TEXTLIST TL_E_CTRL_XPU
  0 = 'XTS_CMD_NULL'
  10 = 'XTS_CMD_INIT'
  30 = 'XTS_IDLE'
   = ''
END_TEXTLIST

(* stored: Version 1.1.0.1, ProductVersion 3.1.4026.18
   TextList TL_E_CTRL_XPU: Id {c1fed775-6cd0-48f3-a5ae-ec8519eac0fa} *)
